TYPE ST_OPCUA :
STRUCT	
	nMyNumber : INT;
	bEnable : BOOL;
	sMessage : STRING;
END_STRUCT
END_TYPE

(* stored: Version 1.1.0.1, ProductVersion 3.1.4024.12
   DUT ST_OPCUA: Id {218a020a-9415-497b-a412-86279d355eab} *)
